{attribute 'GeneratedUsingTerminal: KL3152'}
{attribute addProperty BoxType "KL3152"}
{attribute addProperty Id "Channel_1AT %Q*Channel_03CEAA5E0Channel_2AT %Q*Channel_03CEAA5E0"}
{attribute addProperty CRC "2016972219"}
{attribute addProperty Size "0"}
TYPE KL3152_78388DBB :
STRUCT
	{attribute addProperty Name "Channel_1"}
	Channel_1 : Channel_03CEAA5E;
	{attribute addProperty Name "Channel_2"}
	Channel_2 : Channel_03CEAA5E;
END_STRUCT
END_TYPE

(* stored: Version 1.2.0.0, ProductVersion 3.1.4024.9
   DUT KL3152_78388DBB: Id {e8194423-9131-4422-90c7-2245acfe47bc} *)
